Yaskawa INFORM job: R2_RESET.JBI

/JOB
//NAME R2_RESET
//POS
///NPOS 0,0,0,6,0,0
///TOOL 4
///POSTYPE PULSE
///PULSE
P00017=-183277,-14099,-35332,37951,20141,-66521
///POSTYPE BASE
///RECTAN
///RCONF 0,0,0,0,0,0,0,0,0,0,0,0,0,0,0,0,0,0,0,0,0,0,0,0
P00019=0.000,0.000,2.200,0.0000,0.0000,0.0000
P00021=-1237.685,972.459,470.974,-178.0994,-2.0001,-34.5319
///POSTYPE PULSE
///PULSE
P00027=-163056,-65119,-44243,-3,11,-824
///POSTYPE BASE
///RECTAN
P00028=-1270.000,924.100,955.814,-90.0000,-90.0000,-90.0000
P00029=-1054.000,924.100,968.000,-90.0000,-90.0000,-90.0000
//INST
///DATE 2023/09/11 15:02
///ATTR SC,RW
///GROUP1 RB2
NOP
COMM MOVJ P027
*LOOP
MOVJ P017 PL=0
MOVL P021 PL=0
DOUT OT#(4) ON
MOVL P017 PL=0
WAIT IN#(4)=ON
TIMER T=0.25
SUB P021 P019
DEC I001
TSYNC 1
MOVJ P028 PL=0
TSYNC 2
MOVL P029 PL=0
WAIT OT#(1)=ON
DOUT OT#(4) OFF
TSYNC 3
MOVL P028 PL=0
WAIT IN#(4)=OFF
COMM MOVJ P027
IFTHENEXP I001>=1
	 JUMP *LOOP
ENDIF
SET B003 0
SET B002 1
END
